// TIA Portal V20 export
TYPE "typeIdentRfHmi"
// stored: Access Published
   STRUCT
      selectedRfReader : USInt;   // Reader ID
      selectedAntena : USInt;
      rfReaderId : USInt;   // RF Reader ID
      numberOfRf : USInt;   // Anzahl der RFID Antriebe / Number of used RFIDs
      rfReader : "LSicar_typeIdentInterfaceHmi";   // RF Reader
   END_STRUCT;
END_TYPE
